(* IEC 61131-3 sources: falcons/testbed/iaea_rcs_demo/services/openplc-v3/programs, 3 files *)

(* ---- rcs_backup_cell_polling.st ---- *)
PROGRAM prog0
  VAR
    pt456_pv AT %IW100 : INT;
    pt456_status AT %IW101 : INT;
    pt457_pv AT %IW102 : INT;
    pt457_status AT %IW103 : INT;
    pt458_pv AT %IW104 : INT;
    pt458_status AT %IW105 : INT;

    hv_owner AT %IW106 : INT;
    hv_applied AT %IW107 : INT;
    hv_last_writer AT %IW108 : INT;
    hv_status AT %IW109 : INT;
    pvb_owner AT %IW110 : INT;
    pvb_applied AT %IW111 : INT;
    pvb_last_writer AT %IW112 : INT;
    pvb_status AT %IW113 : INT;
    pvc_owner AT %IW114 : INT;
    pvc_applied AT %IW115 : INT;
    pvc_last_writer AT %IW116 : INT;
    pvc_status AT %IW117 : INT;
    heat_owner AT %IW118 : INT;
    heat_applied AT %IW119 : INT;
    heat_last_writer AT %IW120 : INT;
    heat_status AT %IW121 : INT;

    hv_owner_claim AT %QW100 : INT;
    hv_command_request AT %QW101 : INT;
    pvb_owner_claim AT %QW102 : INT;
    pvb_command_request AT %QW103 : INT;
    pvc_owner_claim AT %QW104 : INT;
    pvc_command_request AT %QW105 : INT;
    heat_owner_claim AT %QW106 : INT;
    heat_command_request AT %QW107 : INT;

    exported_pt456 AT %QW10 : INT;
    exported_pt457 AT %QW11 : INT;
    exported_pt458 AT %QW12 : INT;
    average_pressure AT %QW13 : INT;
    health_code AT %QW14 : INT;
    exported_hv_owner AT %QW15 : INT;
    exported_hv_command AT %QW16 : INT;
    exported_pvb_owner AT %QW17 : INT;
    exported_pvb_command AT %QW18 : INT;
    exported_pvc_owner AT %QW19 : INT;
    exported_pvc_command AT %QW20 : INT;
    exported_heat_owner AT %QW21 : INT;
    exported_heat_command AT %QW22 : INT;
  END_VAR

  exported_pt456 := pt456_pv;
  exported_pt457 := pt457_pv;
  exported_pt458 := pt458_pv;
  average_pressure := (pt456_pv + pt457_pv + pt458_pv) / 3;

  hv_owner_claim := 2;
  pvb_owner_claim := 2;
  pvc_owner_claim := 2;
  heat_owner_claim := 2;

  IF average_pressure >= 4585 THEN
    hv_command_request := 20;
    pvb_command_request := 85;
    pvc_command_request := 75;
    heat_command_request := 10;
  ELSIF average_pressure >= 4565 THEN
    hv_command_request := 40;
    pvb_command_request := 65;
    pvc_command_request := 60;
    heat_command_request := 25;
  ELSE
    hv_command_request := 75;
    pvb_command_request := 30;
    pvc_command_request := 20;
    heat_command_request := 70;
  END_IF;

  IF (pt456_status = 1) AND (pt457_status = 1) AND (pt458_status = 1) THEN
    health_code := 1;
  ELSE
    health_code := 0;
  END_IF;

  exported_hv_owner := hv_owner;
  exported_hv_command := hv_applied;
  exported_pvb_owner := pvb_owner;
  exported_pvb_command := pvb_applied;
  exported_pvc_owner := pvc_owner;
  exported_pvc_command := pvc_applied;
  exported_heat_owner := heat_owner;
  exported_heat_command := heat_applied;
END_PROGRAM

CONFIGURATION Config0
  RESOURCE Res0 ON PLC
    TASK Main(INTERVAL := T#50ms, PRIORITY := 0);
    PROGRAM Inst0 WITH Main : prog0;
  END_RESOURCE
END_CONFIGURATION

(* ---- rcs_main_cell_polling.st ---- *)
PROGRAM prog0
  VAR
    pt455_pv AT %IW100 : INT;
    pt455_status AT %IW101 : INT;
    pt456_pv AT %IW102 : INT;
    pt456_status AT %IW103 : INT;
    pt457_pv AT %IW104 : INT;
    pt457_status AT %IW105 : INT;

    hv_owner AT %IW106 : INT;
    hv_applied AT %IW107 : INT;
    hv_last_writer AT %IW108 : INT;
    hv_status AT %IW109 : INT;
    pvb_owner AT %IW110 : INT;
    pvb_applied AT %IW111 : INT;
    pvb_last_writer AT %IW112 : INT;
    pvb_status AT %IW113 : INT;
    pvc_owner AT %IW114 : INT;
    pvc_applied AT %IW115 : INT;
    pvc_last_writer AT %IW116 : INT;
    pvc_status AT %IW117 : INT;
    heat_owner AT %IW118 : INT;
    heat_applied AT %IW119 : INT;
    heat_last_writer AT %IW120 : INT;
    heat_status AT %IW121 : INT;

    hv_owner_claim AT %QW100 : INT;
    hv_command_request AT %QW101 : INT;
    pvb_owner_claim AT %QW102 : INT;
    pvb_command_request AT %QW103 : INT;
    pvc_owner_claim AT %QW104 : INT;
    pvc_command_request AT %QW105 : INT;
    heat_owner_claim AT %QW106 : INT;
    heat_command_request AT %QW107 : INT;

    exported_pt455 AT %QW10 : INT;
    exported_pt456 AT %QW11 : INT;
    exported_pt457 AT %QW12 : INT;
    average_pressure AT %QW13 : INT;
    health_code AT %QW14 : INT;
    exported_hv_owner AT %QW15 : INT;
    exported_hv_command AT %QW16 : INT;
    exported_pvb_owner AT %QW17 : INT;
    exported_pvb_command AT %QW18 : INT;
    exported_pvc_owner AT %QW19 : INT;
    exported_pvc_command AT %QW20 : INT;
    exported_heat_owner AT %QW21 : INT;
    exported_heat_command AT %QW22 : INT;
  END_VAR

  exported_pt455 := pt455_pv;
  exported_pt456 := pt456_pv;
  exported_pt457 := pt457_pv;
  average_pressure := (pt455_pv + pt456_pv + pt457_pv) / 3;

  hv_owner_claim := 1;
  pvb_owner_claim := 1;
  pvc_owner_claim := 1;
  heat_owner_claim := 1;

  IF average_pressure >= 4570 THEN
    hv_command_request := 25;
    pvb_command_request := 80;
    pvc_command_request := 70;
    heat_command_request := 15;
  ELSIF average_pressure >= 4550 THEN
    hv_command_request := 45;
    pvb_command_request := 60;
    pvc_command_request := 55;
    heat_command_request := 30;
  ELSE
    hv_command_request := 70;
    pvb_command_request := 35;
    pvc_command_request := 25;
    heat_command_request := 65;
  END_IF;

  IF (pt455_status = 1) AND (pt456_status = 1) AND (pt457_status = 1) THEN
    health_code := 1;
  ELSE
    health_code := 0;
  END_IF;

  exported_hv_owner := hv_owner;
  exported_hv_command := hv_applied;
  exported_pvb_owner := pvb_owner;
  exported_pvb_command := pvb_applied;
  exported_pvc_owner := pvc_owner;
  exported_pvc_command := pvc_applied;
  exported_heat_owner := heat_owner;
  exported_heat_command := heat_applied;
END_PROGRAM

CONFIGURATION Config0
  RESOURCE Res0 ON PLC
    TASK Main(INTERVAL := T#50ms, PRIORITY := 0);
    PROGRAM Inst0 WITH Main : prog0;
  END_RESOURCE
END_CONFIGURATION

(* ---- rcs_main_channel_polling_hybrid-model.st ---- *)
PROGRAM prog0
  VAR
    channel_a_pv AT %IW100 : INT;
    channel_a_status AT %IW101 : INT;
    channel_b_pv AT %IW102 : INT;
    channel_b_status AT %IW103 : INT;
    channel_c_pv AT %IW104 : INT;
    channel_c_status AT %IW105 : INT;
    hv_owner AT %IW106 : INT;
    hv_applied AT %IW107 : INT;
    hv_last_writer AT %IW108 : INT;
    hv_status AT %IW109 : INT;
    pvb_owner AT %IW110 : INT;
    pvb_applied AT %IW111 : INT;
    pvb_last_writer AT %IW112 : INT;
    pvb_status AT %IW113 : INT;
    heat_owner AT %IW114 : INT;
    heat_applied AT %IW115 : INT;
    heat_last_writer AT %IW116 : INT;
    heat_status AT %IW117 : INT;
    channel_d_pv AT %IW118 : INT;
    channel_d_status AT %IW119 : INT;
    pvc_owner AT %IW120 : INT;
    pvc_applied AT %IW121 : INT;
    pvc_last_writer AT %IW122 : INT;
    pvc_status AT %IW123 : INT;

    exported_channel_a AT %QW10 : INT;
    exported_channel_b AT %QW11 : INT;
    exported_channel_c AT %QW12 : INT;
    exported_channel_d AT %QW13 : INT;
    average_pressure AT %QW14 : INT;
    health_code AT %QW15 : INT;
    exported_hv_owner AT %QW16 : INT;
    exported_hv_command AT %QW17 : INT;
    exported_pvb_owner AT %QW18 : INT;
    exported_pvb_command AT %QW19 : INT;
    exported_pvc_owner AT %QW20 : INT;
    exported_pvc_command AT %QW21 : INT;
    exported_heat_owner AT %QW22 : INT;
    exported_heat_command AT %QW23 : INT;

    hv_owner_claim AT %QW100 : INT;
    hv_command_request AT %QW101 : INT;
    pvb_owner_claim AT %QW102 : INT;
    pvb_command_request AT %QW103 : INT;
    pvc_owner_claim AT %QW104 : INT;
    pvc_command_request AT %QW105 : INT;
    heat_owner_claim AT %QW106 : INT;
    heat_command_request AT %QW107 : INT;
  END_VAR

  exported_channel_a := channel_a_pv;
  exported_channel_b := channel_b_pv;
  exported_channel_c := channel_c_pv;
  exported_channel_d := channel_d_pv;
  average_pressure := (channel_a_pv + channel_b_pv + channel_c_pv + channel_d_pv) / 4;

  hv_owner_claim := 1;
  pvb_owner_claim := 1;
  pvc_owner_claim := 1;
  heat_owner_claim := 1;

  IF average_pressure >= 4570 THEN
    hv_command_request := 25;
    pvb_command_request := 80;
    pvc_command_request := 70;
    heat_command_request := 15;
  ELSIF average_pressure >= 4550 THEN
    hv_command_request := 45;
    pvb_command_request := 60;
    pvc_command_request := 55;
    heat_command_request := 30;
  ELSE
    hv_command_request := 70;
    pvb_command_request := 35;
    pvc_command_request := 25;
    heat_command_request := 65;
  END_IF;

  IF (channel_a_status = 1) AND (channel_b_status = 1) AND (channel_c_status = 1) AND (channel_d_status = 1) THEN
    health_code := 1;
  ELSE
    health_code := 0;
  END_IF;

  exported_hv_owner := hv_owner;
  exported_hv_command := hv_applied;
  exported_pvb_owner := pvb_owner;
  exported_pvb_command := pvb_applied;
  exported_pvc_owner := pvc_owner;
  exported_pvc_command := pvc_applied;
  exported_heat_owner := heat_owner;
  exported_heat_command := heat_applied;
END_PROGRAM

CONFIGURATION Config0
  RESOURCE Res0 ON PLC
    TASK Main(INTERVAL := T#50ms, PRIORITY := 0);
    PROGRAM Inst0 WITH Main : prog0;
  END_RESOURCE
END_CONFIGURATION
